PROGRAM MAIN
VAR
END_VAR

END_PROGRAM

(* stored: Version 1.1.0.1
   POU MAIN: Id {d39b804c-062b-4229-ae4b-1e01262b0c9e} *)
